{attribute 'qualified_only'}
VAR_GLOBAL
	mb_Input_Coils      : ARRAY[0..255] OF BOOL; //Modbus coils 32768+
	mb_Output_Coils     : ARRAY[0..255] OF BOOL;
	mb_Input_Registers  : ARRAY[0..255] OF WORD; //Modbus input regs 32768+
	mb_Output_Registers : ARRAY[0..255] OF WORD; //Modbus holding regs 32768+
END_VAR

(* stored: Version 1.1.0.1, ProductVersion 3.1.4026.18
   GVL GVL: Id {1640d6a5-390d-47b4-9771-b7f555c5fe9a} *)
